ABB RAPID module: FunctionsGlobalMod.sysx

MODULE FunctionsGlobalMod(SYSMODULE)



    PROC GripOpen()
        !
    ENDPROC



    PROC GripClose()
        !
    ENDPROC



ENDMODULE
